PROGRAM DatabaseRecord
VAR
	test : FB_MemRingBuffer;
END_VAR

// Database Writing actions
GVL.fbInfluxDBRecorder();

END_PROGRAM

(* stored: Version 1.1.0.1, ProductVersion 3.1.4024.12
   POU DatabaseRecord: Id {08677c20-da58-40c4-913e-93c21a52392f}, SpecialFunc None *)
